Staubli VAL3: JointSpace.dtx

public JointPos jointPos
  [0]
    jointRx jp
public JointVel jointVel
  [0]
    num jv[6]
public JointAccel jointAccel
  [0]
    num ja[6]
public JointForce jointForce
  [0]
    num jf[6]
